% RSLogix 500 project PROJECT8-PID SUBSTITUTION LOGIC.RSS, saved by version 8.30.00.16 %
PROJECT "UNTITLED"    % processor: Bul.1763 MicroLogix 1100 Series B %

PROGRAM FILES
  LAD 2 "MAIN"  4 rungs
  LAD 3 "IO"  3 rungs
  LAD 4 "CTRL"  11 rungs

DATA FILES
  O0 OUTPUT  4 elements
  I1 INPUT  6 elements
  S2 STATUS  66 elements
  B3 BINARY  1 elements
  T4 TIMER  1 elements
  C5 COUNTER  1 elements
  R6 CONTROL  1 elements
  N7 INTEGER  6 elements
  F8 FLOAT  2 elements

LADDER 2 "MAIN"
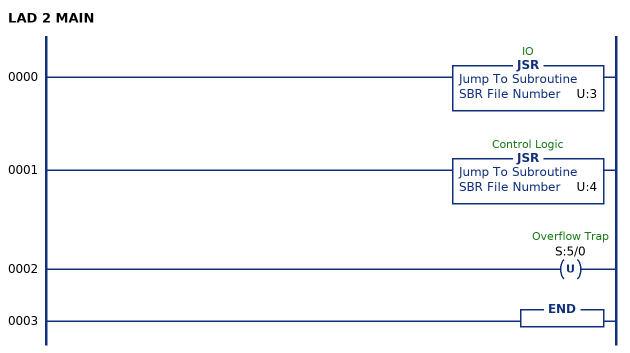
% Rung: 0 %
SOR JSR U:3 EOR
%   U:3  "IO" %
% Rung: 1 %
SOR JSR U:4 EOR
%   U:4  "Control Logic" %
% Rung: 2 %
SOR OTU S:5/0 EOR
%   S:5/0  "Overflow Trap" %
% Rung: 3 %
SOR END EOR

LADDER 3 "IO"
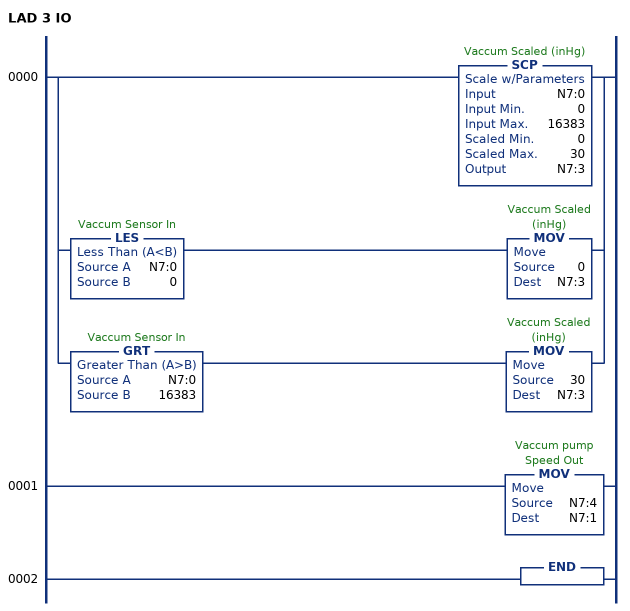
% Rung: 0 %
SOR BST SCP N7:0 0 16383 0 30 N7:3 NXB LES N7:0 0 MOV 0 N7:3 NXB GRT N7:0 16383 MOV 30 N7:3 BND EOR
%   N7:0  "Vaccum Sensor In" %
%   N7:3  "Vaccum Scaled (inHg)" %
% Rung: 1 %
SOR MOV N7:4 N7:1 EOR
%   N7:4  "Calculated Pump Speed" %
%   N7:1  "Vaccum pump Speed Out" %
% Rung: 2 %
SOR END EOR

LADDER 4 "CTRL"
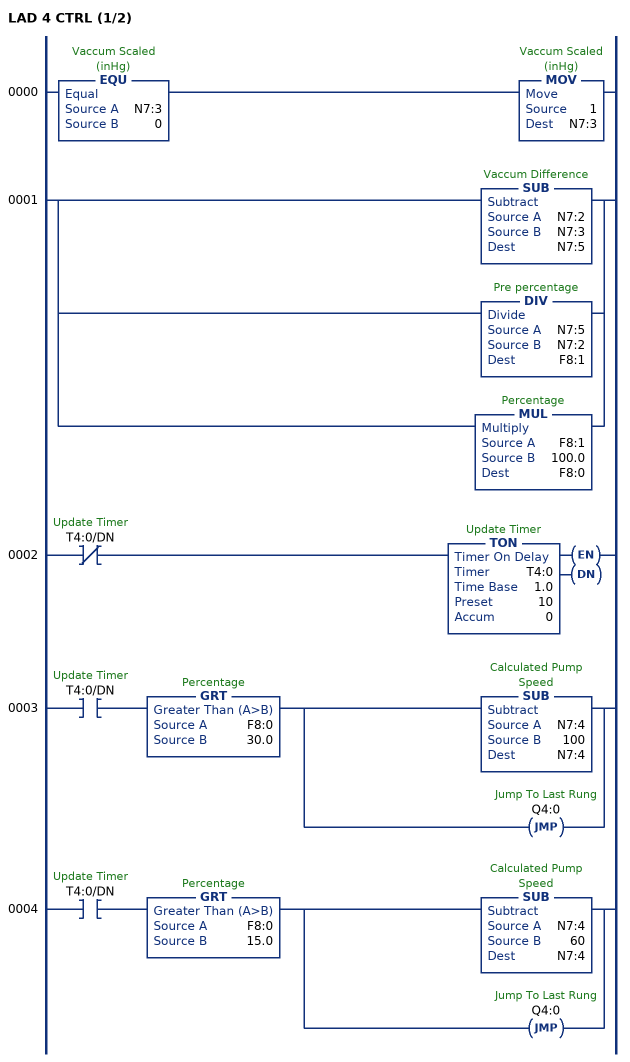
% Rung: 0 %
SOR EQU N7:3 0 MOV 1 N7:3 EOR
%   N7:3  "Vaccum Scaled (inHg)" %
% Rung: 1 %
SOR BST SUB N7:2 N7:3 N7:5 NXB DIV N7:5 N7:2 F8:1 NXB MUL F8:1 100.0 F8:0 BND EOR
%   N7:2  "Setpoint Value" %
%   N7:3  "Vaccum Scaled (inHg)" %
%   N7:5  "Vaccum Difference" %
%   F8:1  "Pre percentage" %
%   F8:0  "Percentage" %
% Rung: 2 %
SOR XIO T4:0/DN TON T4:0 1.0 10 0 EOR
%   T4:0  "Update Timer" %
% Rung: 3 %  % edit flag set %
SOR XIC T4:0/DN GRT F8:0 30.0 BST SUB N7:4 100 N7:4 NXB JMP Q4:0 BND EOR
%   T4:0  "Update Timer" %
%   F8:0  "Percentage" %
%   N7:4  "Calculated Pump Speed" %
%   Q4:0  "Jump To Last Rung" %
% Rung: 4 %  % edit flag set %
SOR XIC T4:0/DN GRT F8:0 15.0 BST SUB N7:4 60 N7:4 NXB JMP Q4:0 BND EOR
%   T4:0  "Update Timer" %
%   F8:0  "Percentage" %
%   N7:4  "Calculated Pump Speed" %
%   Q4:0  "Jump To Last Rung" %

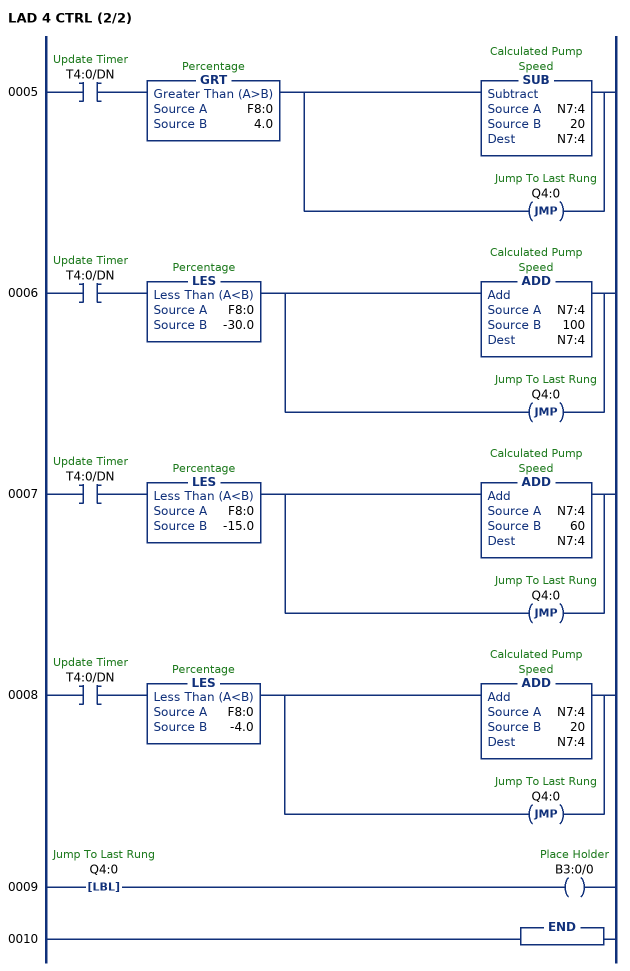
% Rung: 5 %  % edit flag set %
SOR XIC T4:0/DN GRT F8:0 4.0 BST SUB N7:4 20 N7:4 NXB JMP Q4:0 BND EOR
%   T4:0  "Update Timer" %
%   F8:0  "Percentage" %
%   N7:4  "Calculated Pump Speed" %
%   Q4:0  "Jump To Last Rung" %
% Rung: 6 %  % edit flag set %
SOR XIC T4:0/DN LES F8:0 -30.0 BST ADD N7:4 100 N7:4 NXB JMP Q4:0 BND EOR
%   T4:0  "Update Timer" %
%   F8:0  "Percentage" %
%   N7:4  "Calculated Pump Speed" %
%   Q4:0  "Jump To Last Rung" %
% Rung: 7 %  % edit flag set %
SOR XIC T4:0/DN LES F8:0 -15.0 BST ADD N7:4 60 N7:4 NXB JMP Q4:0 BND EOR
%   T4:0  "Update Timer" %
%   F8:0  "Percentage" %
%   N7:4  "Calculated Pump Speed" %
%   Q4:0  "Jump To Last Rung" %
% Rung: 8 %
SOR XIC T4:0/DN LES F8:0 -4.0 BST ADD N7:4 20 N7:4 NXB JMP Q4:0 BND EOR
%   T4:0  "Update Timer" %
%   F8:0  "Percentage" %
%   N7:4  "Calculated Pump Speed" %
%   Q4:0  "Jump To Last Rung" %
% Rung: 9 %
SOR LBL Q4:0 OTE B3:0/0 EOR
%   Q4:0  "Jump To Last Rung" %
%   B3:0/0  "Place Holder" %
% Rung: 10 %
SOR END EOR

DATA TABLE (non-zero values as saved)
DATA T4
% .PRE .ACC %
% T4:0 % 10 0
